{attribute 'GeneratedUsingTerminal: KL9900-0060'}
{attribute addProperty BoxType "KL9900-0060"}
{attribute addProperty Description ""}
{attribute addProperty Physics ""}
{attribute addProperty Id "Channel_1AT %Q*Channel_7D202F580"}
{attribute addProperty CRC "1764799410"}
{attribute addProperty Size "0"}
TYPE KL_6930B3B2 :
STRUCT
	{attribute addProperty Name "Channel_1"}
	Channel_1 : Channel_7D202F58;
END_STRUCT
END_TYPE

(* stored: Version 1.2.0.0, ProductVersion 3.1.4024.11
   DUT KL_6930B3B2: Id {b96b337a-c312-495a-abff-8327c86c3bc9} *)
